KUKA KRL data list: BrakeTestSelfTest.dat

&ACCESS RVO
&REL 1
&PARAM EDITMASK = *
&PARAM TEMPLATE = C:\KRC\Roboter\Template\ExpertVorgabe
DEFDAT BrakeTestSelfTest PUBLIC

INT simulateBrakeVel    = 100
INT simulateBrakeTorque = 50
INT simulateBrakeIndex  = 2

ENDDAT
